PROGRAM MAIN
VAR
	main_fsm	: Main_FSM;
END_VAR

main_fsm();

END_PROGRAM

(* stored: Version 1.1.0.1
   POU MAIN: Id {ee0ed416-3c8e-41d0-b63e-3e0aab4b08ba}, SpecialFunc None *)
